DATA_BLOCK "DB6_ENTIDAD"
{ S7_Optimized_Access := 'FALSE' }
VERSION : 0.1
   STRUCT
      ENT { S7_SetPoint := 'False'} : Array[0.."N_MAX_ENTIDAD"] of "UDT_ZC_PRO_ENTIDAD";
   END_STRUCT;


BEGIN
   ENT[0].Habilitar := TRUE;
   ENT[0].ID := 0;
   ENT[0].Asignacion := 0;
   ENT[0].Estado.Disponible := FALSE;
   ENT[0].Estado.Capturada := FALSE;
   ENT[0].Estado.EnProduccion := FALSE;
   ENT[0].Estado.EnCIP := FALSE;
   ENT[0].Estado.EnSIP := FALSE;
   ENT[0].Estado.EnStandby := FALSE;
   ENT[0].Estado.Limpia := FALSE;
   ENT[0].Estado.Sucia := FALSE;
   ENT[0].Estado.Esterilizada := FALSE;
   ENT[0].Estado.ConProducto := FALSE;
   ENT[0].Estado.ConAgua := FALSE;
   ENT[0].Estado.Vacia := FALSE;
   ENT[0].Estado.Reserva_12 := FALSE;
   ENT[0].Estado.Reserva_13 := FALSE;
   ENT[0].Estado.Reserva_14 := FALSE;
   ENT[0].Estado.Reserva_15 := FALSE;
   ENT[0].Estado.Producto := 0;
   ENT[0].Estado.CodEstado := 0;
   ENT[0].Alarma.Dispositivo := FALSE;
   ENT[0].Alarma.Manual := FALSE;
   ENT[0].Alarma.Reserva_3 := FALSE;
   ENT[0].Alarma.Reserva_4 := FALSE;
   ENT[0].Alarma.Reserva_5 := FALSE;
   ENT[0].Alarma.Reserva_6 := FALSE;
   ENT[0].Alarma.Reserva_7 := FALSE;
   ENT[0].Alarma.Reserva_8 := FALSE;
   ENT[0].Dispositivo[1].Ubicación := 0;
   ENT[0].Dispositivo[1].Tipo := 0;
   ENT[0].Dispositivo[1].Num := 0;
   ENT[0].Dispositivo[2].Ubicación := 0;
   ENT[0].Dispositivo[2].Tipo := 0;
   ENT[0].Dispositivo[2].Num := 0;
   ENT[0].Dispositivo[3].Ubicación := 0;
   ENT[0].Dispositivo[3].Tipo := 0;
   ENT[0].Dispositivo[3].Num := 0;
   ENT[0].Dispositivo[4].Ubicación := 0;
   ENT[0].Dispositivo[4].Tipo := 0;
   ENT[0].Dispositivo[4].Num := 0;
   ENT[0].Dispositivo[5].Ubicación := 0;
   ENT[0].Dispositivo[5].Tipo := 0;
   ENT[0].Dispositivo[5].Num := 0;
   ENT[1].Habilitar := TRUE;
   ENT[1].ID := 1;
   ENT[1].Asignacion := 0;
   ENT[1].Estado.Disponible := TRUE;
   ENT[1].Estado.Capturada := FALSE;
   ENT[1].Estado.EnProduccion := FALSE;
   ENT[1].Estado.EnCIP := FALSE;
   ENT[1].Estado.EnSIP := FALSE;
   ENT[1].Estado.EnStandby := FALSE;
   ENT[1].Estado.Limpia := TRUE;
   ENT[1].Estado.Sucia := FALSE;
   ENT[1].Estado.Esterilizada := FALSE;
   ENT[1].Estado.ConProducto := FALSE;
   ENT[1].Estado.ConAgua := FALSE;
   ENT[1].Estado.Vacia := FALSE;
   ENT[1].Estado.Reserva_12 := FALSE;
   ENT[1].Estado.Reserva_13 := FALSE;
   ENT[1].Estado.Reserva_14 := FALSE;
   ENT[1].Estado.Reserva_15 := FALSE;
   ENT[1].Estado.Producto := 0;
   ENT[1].Estado.CodEstado := 11000;
   ENT[1].Alarma.Dispositivo := FALSE;
   ENT[1].Alarma.Manual := FALSE;
   ENT[1].Alarma.Reserva_3 := FALSE;
   ENT[1].Alarma.Reserva_4 := FALSE;
   ENT[1].Alarma.Reserva_5 := FALSE;
   ENT[1].Alarma.Reserva_6 := FALSE;
   ENT[1].Alarma.Reserva_7 := FALSE;
   ENT[1].Alarma.Reserva_8 := FALSE;
   ENT[1].Dispositivo[1].Ubicación := 0;
   ENT[1].Dispositivo[1].Tipo := 0;
   ENT[1].Dispositivo[1].Num := 0;
   ENT[1].Dispositivo[2].Ubicación := 0;
   ENT[1].Dispositivo[2].Tipo := 0;
   ENT[1].Dispositivo[2].Num := 0;
   ENT[1].Dispositivo[3].Ubicación := 0;
   ENT[1].Dispositivo[3].Tipo := 0;
   ENT[1].Dispositivo[3].Num := 0;
   ENT[1].Dispositivo[4].Ubicación := 0;
   ENT[1].Dispositivo[4].Tipo := 0;
   ENT[1].Dispositivo[4].Num := 0;
   ENT[1].Dispositivo[5].Ubicación := 0;
   ENT[1].Dispositivo[5].Tipo := 0;
   ENT[1].Dispositivo[5].Num := 0;

END_DATA_BLOCK

